// LS Electric XG5000 project: PLC Trancemit PC Recive
// PLC LSPLC

PROGRAM NewProgram (task: 스캔 프로그램)

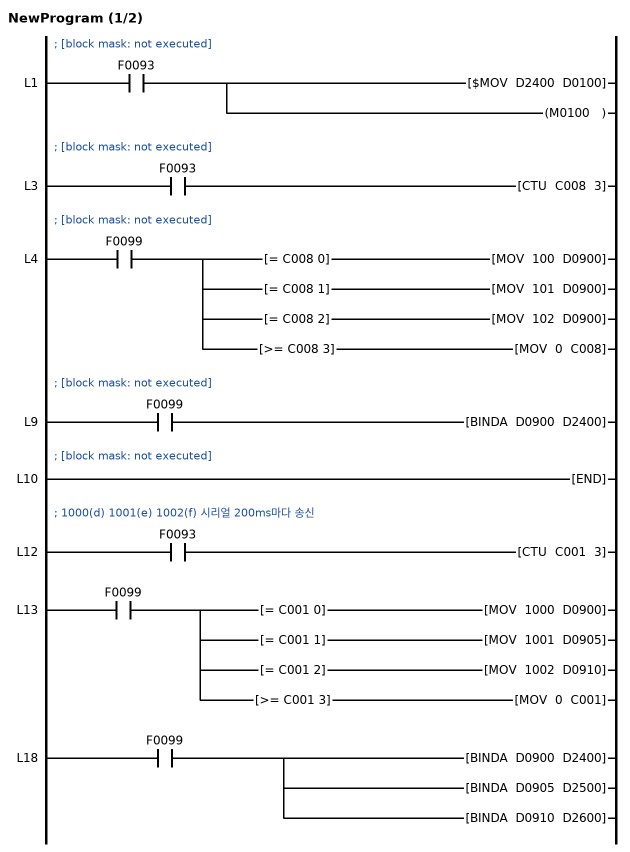
; L1 (block mask: not executed)
LOAD      F0093
$MOV      D2400 D0100
OUT       M0100
; L3 (block mask: not executed)
LOAD      F0093
CTU       C008 3
; L4 (block mask: not executed)
LOAD      F0099
MPUSH
AND=      C008 0
MOV       100 D0900
MLOAD
AND=      C008 1
MOV       101 D0900
MLOAD
AND=      C008 2
MOV       102 D0900
MPOP
AND>=     C008 3
MOV       0 C008
; L9 (block mask: not executed)
LOAD      F0099
BINDA     D0900 D2400
; L10 (block mask: not executed)
END
// 1000(d) 1001(e) 1002(f) 시리얼 200ms마다 송신
; L12
LOAD      F0093
CTU       C001 3
; L13
LOAD      F0099
MPUSH
AND=      C001 0
MOV       1000 D0900
MLOAD
AND=      C001 1
MOV       1001 D0905
MLOAD
AND=      C001 2
MOV       1002 D0910
MPOP
AND>=     C001 3
MOV       0 C001
; L18
LOAD      F0099
BINDA     D0900 D2400
BINDA     D0905 D2500
BINDA     D0910 D2600

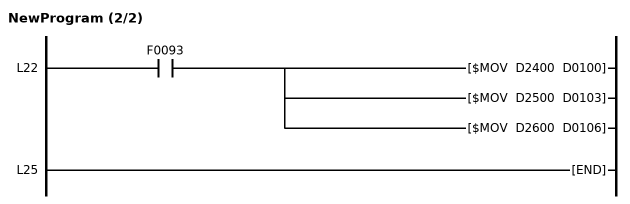
; L22
LOAD      F0093
$MOV      D2400 D0100
$MOV      D2500 D0103
$MOV      D2600 D0106
; L25
END